// TIA Portal V18 export
// export: Created 2026-06-21T12:15:02Z, ExportSetting WithDefaults
PlcWatchTable "WT_PLC2_Main_Sequence"
  PlcWatchTableEntry "HMI_Sim_Mode"
  PlcWatchTableEntry "HMI_Use_Sim_Input_PLC2"
  PlcWatchTableEntry "PLC2_State"
  PlcWatchTableEntry "PLC2_Loi_Tong"
  PlcWatchTableEntry "FQ3210_Bon3_HMI"
  PlcWatchTableEntry "LT3213_Bon3_HMI"
  PlcWatchTableEntry "FQ3215_Bon4_HMI"
  PlcWatchTableEntry "LT3218_Bon4_HMI"
  PlcWatchTableEntry "TT3219_Bon4_HMI"
  PlcWatchTableEntry "V3240_Nuoc_Bon3"
  PlcWatchTableEntry "AGTR3262_Khuay_Bon3"
  PlcWatchTableEntry "V3245_Nuoc_Bon4"
  PlcWatchTableEntry "CV3216_Hoi_Bon4"
  PlcWatchTableEntry "AGTR3263_Khuay_Bon4"
  PlcWatchTableEntry "AGTR3263_Dao_Chieu"
  PlcWatchTableEntry "Pump3265_Chuyen_Nhanh2"
  PlcWatchTableEntry "PLC2_Me_Nhanh2_Hoan_Thanh"
  PlcWatchTableEntry "PLC2_Xa_Bon4_Xong"
  PlcWatchTableEntry "HMI_Anim_Bon3_Frame"
  PlcWatchTableEntry "HMI_Anim_Bon4_Frame"
